SUBAPPLICATION Uebung_040 (* Lauflicht 8 *)
  (* Standard: 61499-2 *)
  (* Version 1.0, 2023-10-23, franz *)
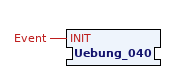
  EVENT_INPUT
    INIT;
  END_EVENT
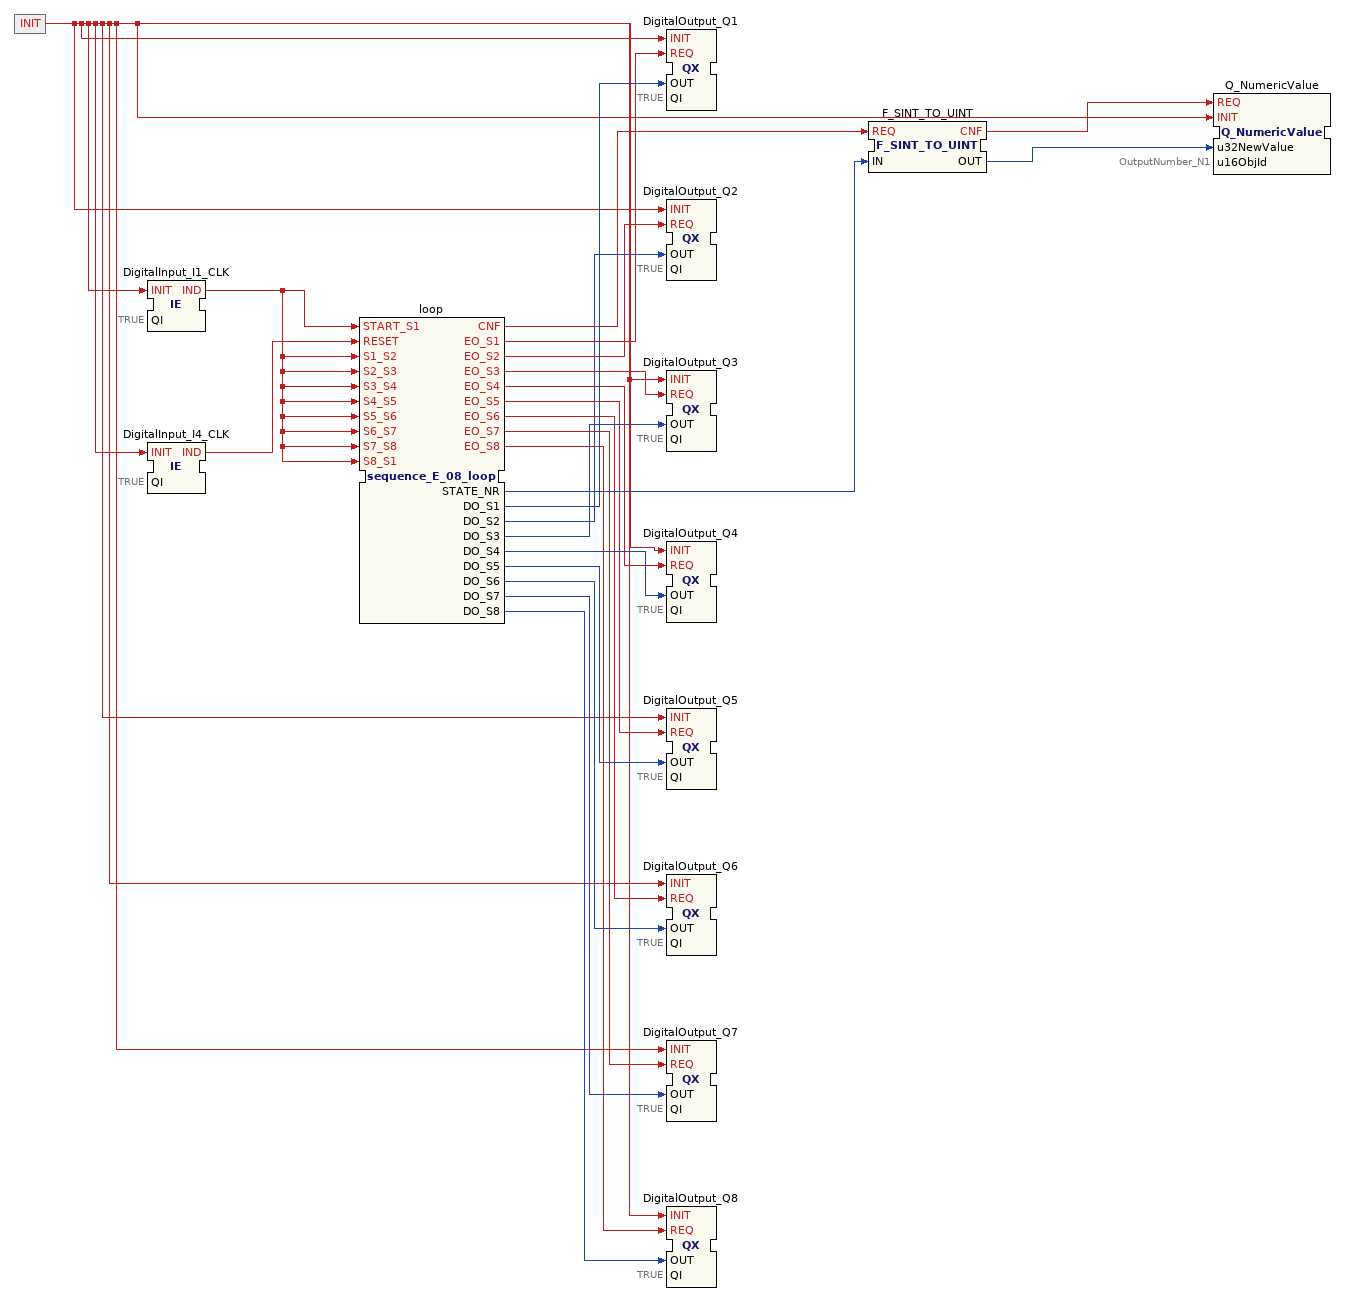
  FBS
    DigitalOutput_Q1 : QX(QI := TRUE);
    DigitalOutput_Q2 : QX(QI := TRUE);
    DigitalOutput_Q3 : QX(QI := TRUE);
    DigitalOutput_Q4 : QX(QI := TRUE);
    DigitalInput_I1_CLK : IE(QI := TRUE);
    DigitalInput_I4_CLK : IE(QI := TRUE);
    DigitalOutput_Q5 : QX(QI := TRUE);
    DigitalOutput_Q6 : QX(QI := TRUE);
    DigitalOutput_Q7 : QX(QI := TRUE);
    DigitalOutput_Q8 : QX(QI := TRUE);
    Q_NumericValue : Q_NumericValue(u16ObjId := OutputNumber_N1);
    F_SINT_TO_UINT : F_SINT_TO_UINT;
    loop : sequence_E_08_loop;
  END_FBS
  EVENT_CONNECTIONS
    INIT TO DigitalOutput_Q4.INIT;
    INIT TO DigitalOutput_Q3.INIT;
    INIT TO DigitalOutput_Q2.INIT;
    INIT TO DigitalOutput_Q1.INIT;
    INIT TO DigitalInput_I1_CLK.INIT;
    INIT TO DigitalInput_I4_CLK.INIT;
    INIT TO DigitalOutput_Q5.INIT;
    INIT TO DigitalOutput_Q6.INIT;
    INIT TO DigitalOutput_Q7.INIT;
    INIT TO DigitalOutput_Q8.INIT;
    F_SINT_TO_UINT.CNF TO Q_NumericValue.REQ;
    INIT TO Q_NumericValue.INIT;
    DigitalInput_I1_CLK.IND TO loop.START_S1;
    DigitalInput_I4_CLK.IND TO loop.RESET;
    loop.CNF TO F_SINT_TO_UINT.REQ;
    loop.EO_S1 TO DigitalOutput_Q1.REQ;
    loop.EO_S2 TO DigitalOutput_Q2.REQ;
    loop.EO_S3 TO DigitalOutput_Q3.REQ;
    loop.EO_S4 TO DigitalOutput_Q4.REQ;
    loop.EO_S5 TO DigitalOutput_Q5.REQ;
    loop.EO_S6 TO DigitalOutput_Q6.REQ;
    loop.EO_S7 TO DigitalOutput_Q7.REQ;
    loop.EO_S8 TO DigitalOutput_Q8.REQ;
    DigitalInput_I1_CLK.IND TO loop.S1_S2;
    DigitalInput_I1_CLK.IND TO loop.S2_S3;
    DigitalInput_I1_CLK.IND TO loop.S3_S4;
    DigitalInput_I1_CLK.IND TO loop.S4_S5;
    DigitalInput_I1_CLK.IND TO loop.S5_S6;
    DigitalInput_I1_CLK.IND TO loop.S6_S7;
    DigitalInput_I1_CLK.IND TO loop.S7_S8;
    DigitalInput_I1_CLK.IND TO loop.S8_S1;
  END_CONNECTIONS
  DATA_CONNECTIONS
    F_SINT_TO_UINT.OUT TO Q_NumericValue.u32NewValue;
    loop.STATE_NR TO F_SINT_TO_UINT.IN;
    loop.DO_S1 TO DigitalOutput_Q1.OUT;
    loop.DO_S2 TO DigitalOutput_Q2.OUT;
    loop.DO_S3 TO DigitalOutput_Q3.OUT;
    loop.DO_S4 TO DigitalOutput_Q4.OUT;
    loop.DO_S5 TO DigitalOutput_Q5.OUT;
    loop.DO_S6 TO DigitalOutput_Q6.OUT;
    loop.DO_S7 TO DigitalOutput_Q7.OUT;
    loop.DO_S8 TO DigitalOutput_Q8.OUT;
  END_CONNECTIONS
END_SUBAPPLICATION
